FUNCTION_BLOCK PUBLIC DT_TO_TestSuite EXTENDS TcUnit.FB_TestSuite
VAR
END_VAR

Check_DT_TO_BOOL_Max();
Check_DT_TO_BOOL_Min();
Check_DT_TO_BYTE_Max();
Check_DT_TO_BYTE_Min();
Check_DT_TO_BYTE_TooHigh();
Check_DT_TO_WORD_Max();
Check_DT_TO_WORD_Min();
Check_DT_TO_WORD_TooHigh();
Check_DT_TO_DWORD_Max();
Check_DT_TO_DWORD_Min();
Check_DT_TO_LWORD_Max();
Check_DT_TO_LWORD_Min();
Check_DT_TO_SINT_Max();
Check_DT_TO_SINT_Min();
Check_DT_TO_SINT_TooHigh();
Check_DT_TO_INT_Max();
Check_DT_TO_INT_Min();
Check_DT_TO_INT_TooHigh();
Check_DT_TO_DINT_Max();
Check_DT_TO_DINT_Min();
Check_DT_TO_DINT_TooHigh();
Check_DT_TO_LINT_Max();
Check_DT_TO_LINT_Min();
Check_DT_TO_USINT_Max();
Check_DT_TO_USINT_Min();
Check_DT_TO_USINT_TooHigh();
Check_DT_TO_UINT_Max();
Check_DT_TO_UINT_Min();
Check_DT_TO_UINT_TooHigh();
Check_DT_TO_UDINT_Max();
Check_DT_TO_UDINT_Min();
Check_DT_TO_ULINT_Max();
Check_DT_TO_ULINT_Min();
Check_DT_TO_REAL_Max();
Check_DT_TO_REAL_Min();
Check_DT_TO_LREAL_Max();
Check_DT_TO_LREAL_Min();
Check_DT_TO_TIME_Max();
Check_DT_TO_TIME_Min();
Check_DT_TO_TIME_TooHigh();
Check_DT_TO_TOD_Max();
Check_DT_TO_TOD_Min();
Check_DT_TO_TOD_TooHigh();
Check_DT_TO_DATE_Max();
Check_DT_TO_DATE_Min();
Check_DT_TO_DT_Max();
Check_DT_TO_DT_Min();
Check_DT_TO_STRING_Max();
Check_DT_TO_STRING_Min();

METHOD PUBLIC Check_DT_TO_BOOL_Min
VAR
	value : DT := DatatypeLimits.DT_MIN_VALUE;
	actual : BOOL;
	converted : BOOL;
	equal : BOOL;
END_VAR
TEST('Check_DT_TO_BOOL_Min');

// @TEST-RUN
converted := TryConvert_DT_TO_Destination(value, actual);
equal := actual = DT_TO_BOOL(value);

// @TEST-ASSERT
AssertTrue(Condition := equal, Message := 'Did not convert DT to BOOL correctly');
AssertTrue(Condition := converted, Message := 'Did not report DT to BOOL conversion was successful');

TEST_FINISHED();
END_METHOD

METHOD PUBLIC Check_DT_TO_BOOL_Max
VAR
	value : DT := DatatypeLimits.DT_MAX_VALUE;
	actual : BOOL;
	converted : BOOL;
	equal : BOOL;
END_VAR
TEST('Check_DT_TO_BOOL_Max');

// @TEST-RUN
converted := TryConvert_DT_TO_Destination(value, actual);
equal := actual = DT_TO_BOOL(value);

// @TEST-ASSERT
AssertTrue(Condition := equal, Message := 'Did not convert DT to BOOL correctly');
AssertTrue(Condition := converted, Message := 'Did not report DT to BOOL conversion was successful');

TEST_FINISHED();
END_METHOD

METHOD PUBLIC Check_DT_TO_BYTE_Min
VAR
	value : DT := DatatypeLimits.DT_MIN_VALUE;
	actual : BYTE;
	converted : BOOL;
	equal : BOOL;
END_VAR
TEST('Check_DT_TO_BYTE_Min');

// @TEST-RUN
converted := TryConvert_DT_TO_Destination(value, actual);
equal := actual = DT_TO_BYTE(value);

// @TEST-ASSERT
AssertTrue(Condition := equal, Message := 'Did not convert DT to BYTE correctly');
AssertTrue(Condition := converted, Message := 'Did not report DT to BYTE conversion was successful');

TEST_FINISHED();
END_METHOD

METHOD PUBLIC Check_DT_TO_BYTE_TooHigh
VAR
	value : DT := DatatypeLimits.DT_MAX_VALUE;
	actual : BYTE;
	converted : BOOL;
END_VAR
TEST('Check_DT_TO_BYTE_TooHigh');

// @TEST-RUN
converted := TryConvert_DT_TO_Destination(value, actual);

// @TEST-ASSERT
AssertFalse(Condition := converted, Message := 'Did not report DT to BYTE conversion was prevented');

TEST_FINISHED();
END_METHOD

METHOD PUBLIC Check_DT_TO_BYTE_Max
VAR
	value : DT := DatatypeLimits.MAX_VALUE_OF_DT_WHICH_CAN_BE_HELD_IN_A_BYTE;
	actual : BYTE;
	converted : BOOL;
	equal : BOOL;
END_VAR
TEST('Check_DT_TO_BYTE_Max');

// @TEST-RUN
converted := TryConvert_DT_TO_Destination(value, actual);
equal := actual = DT_TO_BYTE(value);

// @TEST-ASSERT
AssertTrue(Condition := equal, Message := 'Did not convert DT to BYTE correctly');
AssertTrue(Condition := converted, Message := 'Did not report DT to BYTE conversion was successful');

TEST_FINISHED();
END_METHOD

METHOD PUBLIC Check_DT_TO_DATE_Min
VAR
	value : DT := DatatypeLimits.DT_MIN_VALUE;
	actual : DATE;
	converted : BOOL;
	equal : BOOL;
END_VAR
TEST('Check_DT_TO_DATE_Min');

// @TEST-RUN
converted := TryConvert_DT_TO_Destination(value, actual);
equal := actual = DT_TO_DATE(value);

// @TEST-ASSERT
AssertTrue(Condition := equal, Message := 'Did not convert DT to DATE correctly');
AssertTrue(Condition := converted, Message := 'Did not report DT to DATE conversion was successful');

TEST_FINISHED();
END_METHOD

METHOD PUBLIC Check_DT_TO_DATE_Max
VAR
	value : DT := DatatypeLimits.DT_MAX_VALUE;
	actual : DATE;
	converted : BOOL;
	equal : BOOL;
END_VAR
TEST('Check_DT_TO_DATE_Max');

// @TEST-RUN
converted := TryConvert_DT_TO_Destination(value, actual);
equal := actual = DT_TO_DATE(value);

// @TEST-ASSERT
AssertTrue(Condition := equal, Message := 'Did not convert DT to DATE correctly');
AssertTrue(Condition := converted, Message := 'Did not report DT to DATE conversion was successful');

TEST_FINISHED();
END_METHOD

METHOD PUBLIC Check_DT_TO_DINT_Min
VAR
	value : DT := DatatypeLimits.DT_MIN_VALUE;
	actual : DINT;
	converted : BOOL;
	equal : BOOL;
END_VAR
TEST('Check_DT_TO_DINT_Min');

// @TEST-RUN
converted := TryConvert_DT_TO_Destination(value, actual);
equal := actual = DT_TO_DINT(value);

// @TEST-ASSERT
AssertTrue(Condition := equal, Message := 'Did not convert DT to DINT correctly');
AssertTrue(Condition := converted, Message := 'Did not report DT to DINT conversion was successful');

TEST_FINISHED();
END_METHOD

METHOD PUBLIC Check_DT_TO_DINT_TooHigh
VAR
	value : DT := DatatypeLimits.DT_MAX_VALUE;
	actual : DINT;
	converted : BOOL;
END_VAR
TEST('Check_DT_TO_DINT_TooHigh');

// @TEST-RUN
converted := TryConvert_DT_TO_Destination(value, actual);

// @TEST-ASSERT
AssertFalse(Condition := converted, Message := 'Did not report DT to DINT conversion was prevented');

TEST_FINISHED();
END_METHOD

METHOD PUBLIC Check_DT_TO_DINT_Max
VAR
	value : DT := DatatypeLimits.MAX_VALUE_OF_DT_WHICH_CAN_BE_HELD_IN_A_DINT;
	actual : DINT;
	converted : BOOL;
	equal : BOOL;
END_VAR
TEST('Check_DT_TO_DINT_Max');

// @TEST-RUN
converted := TryConvert_DT_TO_Destination(value, actual);
equal := actual = DT_TO_DINT(value);

// @TEST-ASSERT
AssertTrue(Condition := equal, Message := 'Did not convert DT to DINT correctly');
AssertTrue(Condition := converted, Message := 'Did not report DT to DINT conversion was successful');

TEST_FINISHED();
END_METHOD

METHOD PUBLIC Check_DT_TO_DT_Min
VAR
	value : DT := DatatypeLimits.DT_MIN_VALUE;
	actual : DT;
	converted : BOOL;
	equal : BOOL;
END_VAR
TEST('Check_DT_TO_DT_Min');

// @TEST-RUN
converted := TryConvert_DT_TO_Destination(value, actual);
equal := actual = value;

// @TEST-ASSERT
AssertTrue(Condition := equal, Message := 'Did not convert DT to DT correctly');
AssertTrue(Condition := converted, Message := 'Did not report DT to DT conversion was successful');

TEST_FINISHED();
END_METHOD

METHOD PUBLIC Check_DT_TO_DT_Max
VAR
	value : DT := DatatypeLimits.DT_MAX_VALUE;
	actual : DT;
	converted : BOOL;
	equal : BOOL;
END_VAR
TEST('Check_DT_TO_DT_Max');

// @TEST-RUN
converted := TryConvert_DT_TO_Destination(value, actual);
equal := actual = value;

// @TEST-ASSERT
AssertTrue(Condition := equal, Message := 'Did not convert DT to DT correctly');
AssertTrue(Condition := converted, Message := 'Did not report DT to DT conversion was successful');

TEST_FINISHED();
END_METHOD

METHOD PUBLIC Check_DT_TO_DWORD_Min
VAR
	value : DT := DatatypeLimits.DT_MIN_VALUE;
	actual : DWORD;
	converted : BOOL;
	equal : BOOL;
END_VAR
TEST('Check_DT_TO_DWORD_Min');

// @TEST-RUN
converted := TryConvert_DT_TO_Destination(value, actual);
equal := actual = DT_TO_DWORD(value);

// @TEST-ASSERT
AssertTrue(Condition := equal, Message := 'Did not convert DT to DWORD correctly');
AssertTrue(Condition := converted, Message := 'Did not report DT to DWORD conversion was successful');

TEST_FINISHED();
END_METHOD

METHOD PUBLIC Check_DT_TO_DWORD_Max
VAR
	value : DT := DatatypeLimits.DT_MAX_VALUE;
	actual : DWORD;
	converted : BOOL;
	equal : BOOL;
END_VAR
TEST('Check_DT_TO_DWORD_Max');

// @TEST-RUN
converted := TryConvert_DT_TO_Destination(value, actual);
equal := actual = DT_TO_DWORD(value);

// @TEST-ASSERT
AssertTrue(Condition := equal, Message := 'Did not convert DT to DWORD correctly');
AssertTrue(Condition := converted, Message := 'Did not report DT to DWORD conversion was successful');

TEST_FINISHED();
END_METHOD

METHOD PUBLIC Check_DT_TO_INT_Min
VAR
	value : DT := DatatypeLimits.DT_MIN_VALUE;
	actual : INT;
	converted : BOOL;
	equal : BOOL;
END_VAR
TEST('Check_DT_TO_INT_Min');

// @TEST-RUN
converted := TryConvert_DT_TO_Destination(value, actual);
equal := actual = DT_TO_INT(value);

// @TEST-ASSERT
AssertTrue(Condition := equal, Message := 'Did not convert DT to INT correctly');
AssertTrue(Condition := converted, Message := 'Did not report DT to INT conversion was successful');

TEST_FINISHED();
END_METHOD

METHOD PUBLIC Check_DT_TO_INT_TooHigh
VAR
	value : DT := DatatypeLimits.DT_MAX_VALUE;
	actual : INT;
	converted : BOOL;
END_VAR
TEST('Check_DT_TO_INT_TooHigh');

// @TEST-RUN
converted := TryConvert_DT_TO_Destination(value, actual);

// @TEST-ASSERT
AssertFalse(Condition := converted, Message := 'Did not report DT to INT conversion was prevented');

TEST_FINISHED();
END_METHOD

METHOD PUBLIC Check_DT_TO_INT_Max
VAR
	value : DT := DatatypeLimits.MAX_VALUE_OF_DT_WHICH_CAN_BE_HELD_IN_A_INT;
	actual : INT;
	converted : BOOL;
	equal : BOOL;
END_VAR
TEST('Check_DT_TO_INT_Max');

// @TEST-RUN
converted := TryConvert_DT_TO_Destination(value, actual);
equal := actual = DT_TO_INT(value);

// @TEST-ASSERT
AssertTrue(Condition := equal, Message := 'Did not convert DT to INT correctly');
AssertTrue(Condition := converted, Message := 'Did not report DT to INT conversion was successful');

TEST_FINISHED();
END_METHOD

METHOD PUBLIC Check_DT_TO_LINT_Min
VAR
	value : DT := DatatypeLimits.DT_MIN_VALUE;
	actual : LINT;
	converted : BOOL;
	equal : BOOL;
END_VAR
TEST('Check_DT_TO_LINT_Min');

// @TEST-RUN
converted := TryConvert_DT_TO_Destination(value, actual);
equal := actual = DT_TO_LINT(value);

// @TEST-ASSERT
AssertTrue(Condition := equal, Message := 'Did not convert DT to LINT correctly');
AssertTrue(Condition := converted, Message := 'Did not report DT to LINT conversion was successful');

TEST_FINISHED();
END_METHOD

METHOD PUBLIC Check_DT_TO_LINT_Max
VAR
	value : DT := DatatypeLimits.DT_MAX_VALUE;
	actual : LINT;
	converted : BOOL;
	equal : BOOL;
END_VAR
TEST('Check_DT_TO_LINT_Max');

// @TEST-RUN
converted := TryConvert_DT_TO_Destination(value, actual);
equal := actual = DT_TO_LINT(value);

// @TEST-ASSERT
AssertTrue(Condition := equal, Message := 'Did not convert DT to LINT correctly');
AssertTrue(Condition := converted, Message := 'Did not report DT to LINT conversion was successful');

TEST_FINISHED();
END_METHOD

METHOD PUBLIC Check_DT_TO_LREAL_Min
VAR
	value : DT := DatatypeLimits.DT_MIN_VALUE;
	actual : LREAL;
	converted : BOOL;
	equal : BOOL;
END_VAR
TEST('Check_DT_TO_LREAL_Min');

// @TEST-RUN
converted := TryConvert_DT_TO_Destination(value, actual);
equal := actual = DT_TO_LREAL(value);

// @TEST-ASSERT
AssertTrue(Condition := equal, Message := 'Did not convert DT to LREAL correctly');
AssertTrue(Condition := converted, Message := 'Did not report DT to LREAL conversion was successful');

TEST_FINISHED();
END_METHOD

METHOD PUBLIC Check_DT_TO_LREAL_Max
VAR
	value : DT := DatatypeLimits.DT_MAX_VALUE;
	actual : LREAL;
	converted : BOOL;
	equal : BOOL;
END_VAR
TEST('Check_DT_TO_LREAL_Max');

// @TEST-RUN
converted := TryConvert_DT_TO_Destination(value, actual);
equal := actual = DT_TO_LREAL(value);

// @TEST-ASSERT
AssertTrue(Condition := equal, Message := 'Did not convert DT to LREAL correctly');
AssertTrue(Condition := converted, Message := 'Did not report DT to LREAL conversion was successful');

TEST_FINISHED();
END_METHOD

METHOD PUBLIC Check_DT_TO_LWORD_Min
VAR
	value : DT := DatatypeLimits.DT_MIN_VALUE;
	actual : LWORD;
	converted : BOOL;
	equal : BOOL;
END_VAR
TEST('Check_DT_TO_LWORD_Min');

// @TEST-RUN
converted := TryConvert_DT_TO_Destination(value, actual);
equal := actual = DT_TO_LWORD(value);

// @TEST-ASSERT
AssertTrue(Condition := equal, Message := 'Did not convert DT to LWORD correctly');
AssertTrue(Condition := converted, Message := 'Did not report DT to LWORD conversion was successful');

TEST_FINISHED();
END_METHOD

METHOD PUBLIC Check_DT_TO_LWORD_Max
VAR
	value : DT := DatatypeLimits.DT_MAX_VALUE;
	actual : LWORD;
	converted : BOOL;
	equal : BOOL;
END_VAR
TEST('Check_DT_TO_LWORD_Max');

// @TEST-RUN
converted := TryConvert_DT_TO_Destination(value, actual);
equal := actual = DT_TO_LWORD(value);

// @TEST-ASSERT
AssertTrue(Condition := equal, Message := 'Did not convert DT to LWORD correctly');
AssertTrue(Condition := converted, Message := 'Did not report DT to LWORD conversion was successful');

TEST_FINISHED();
END_METHOD

METHOD PUBLIC Check_DT_TO_REAL_Min
VAR
	value : DT := DatatypeLimits.DT_MIN_VALUE;
	actual : REAL;
	converted : BOOL;
	equal : BOOL;
END_VAR
TEST('Check_DT_TO_REAL_Min');

// @TEST-RUN
converted := TryConvert_DT_TO_Destination(value, actual);
equal := actual = DT_TO_REAL(value);

// @TEST-ASSERT
AssertTrue(Condition := equal, Message := 'Did not convert DT to REAL correctly');
AssertTrue(Condition := converted, Message := 'Did not report DT to REAL conversion was successful');

TEST_FINISHED();
END_METHOD

METHOD PUBLIC Check_DT_TO_REAL_Max
VAR
	value : DT := DatatypeLimits.DT_MAX_VALUE;
	actual : REAL;
	converted : BOOL;
	equal : BOOL;
END_VAR
TEST('Check_DT_TO_REAL_Max');

// @TEST-RUN
converted := TryConvert_DT_TO_Destination(value, actual);
equal := actual = DT_TO_REAL(value);

// @TEST-ASSERT
AssertTrue(Condition := equal, Message := 'Did not convert DT to REAL correctly');
AssertTrue(Condition := converted, Message := 'Did not report DT to REAL conversion was successful');

TEST_FINISHED();
END_METHOD

METHOD PUBLIC Check_DT_TO_SINT_Min
VAR
	value : DT := DatatypeLimits.DT_MIN_VALUE;
	actual : SINT;
	converted : BOOL;
	equal : BOOL;
END_VAR
TEST('Check_DT_TO_SINT_Min');

// @TEST-RUN
converted := TryConvert_DT_TO_Destination(value, actual);
equal := actual = DT_TO_SINT(value);

// @TEST-ASSERT
AssertTrue(Condition := equal, Message := 'Did not convert DT to SINT correctly');
AssertTrue(Condition := converted, Message := 'Did not report DT to SINT conversion was successful');

TEST_FINISHED();
END_METHOD

METHOD PUBLIC Check_DT_TO_SINT_TooHigh
VAR
	value : DT := DatatypeLimits.DT_MAX_VALUE;
	actual : SINT;
	converted : BOOL;
END_VAR
TEST('Check_DT_TO_SINT_TooHigh');

// @TEST-RUN
converted := TryConvert_DT_TO_Destination(value, actual);

// @TEST-ASSERT
AssertFalse(Condition := converted, Message := 'Did not report DT to SINT conversion was prevented');

TEST_FINISHED();
END_METHOD

METHOD PUBLIC Check_DT_TO_SINT_Max
VAR
	value : DT := DatatypeLimits.MAX_VALUE_OF_DT_WHICH_CAN_BE_HELD_IN_A_SINT;
	actual : SINT;
	converted : BOOL;
	equal : BOOL;
END_VAR
TEST('Check_DT_TO_SINT_Max');

// @TEST-RUN
converted := TryConvert_DT_TO_Destination(value, actual);
equal := actual = DT_TO_SINT(value);

// @TEST-ASSERT
AssertTrue(Condition := equal, Message := 'Did not convert DT to SINT correctly');
AssertTrue(Condition := converted, Message := 'Did not report DT to SINT conversion was successful');

TEST_FINISHED();
END_METHOD

METHOD PUBLIC Check_DT_TO_STRING_Min
VAR
	value : DT := DatatypeLimits.DT_MIN_VALUE;
	actual : STRING;
	converted : BOOL;
	equal : BOOL;
END_VAR
TEST('Check_DT_TO_STRING_Min');

// @TEST-RUN
converted := TryConvert_DT_TO_Destination(value, actual);
equal := actual = DT_TO_STRING(value);

// @TEST-ASSERT
AssertTrue(Condition := equal, Message := 'Did not convert DT to STRING correctly');
AssertTrue(Condition := converted, Message := 'Did not report DT to STRING conversion was successful');

TEST_FINISHED();
END_METHOD

METHOD PUBLIC Check_DT_TO_STRING_Max
VAR
	value : DT := DatatypeLimits.DT_MAX_VALUE;
	actual : STRING;
	converted : BOOL;
	equal : BOOL;
END_VAR
TEST('Check_DT_TO_STRING_Max');

// @TEST-RUN
converted := TryConvert_DT_TO_Destination(value, actual);
equal := actual = DT_TO_STRING(value);

// @TEST-ASSERT
AssertTrue(Condition := equal, Message := 'Did not convert DT to STRING correctly');
AssertTrue(Condition := converted, Message := 'Did not report DT to STRING conversion was successful');

TEST_FINISHED();
END_METHOD

METHOD PUBLIC Check_DT_TO_TIME_Min
VAR
	value : DT := DatatypeLimits.DT_MIN_VALUE;
	actual : TIME;
	converted : BOOL;
	equal : BOOL;
END_VAR
TEST('Check_DT_TO_TIME_Min');

// @TEST-RUN
converted := TryConvert_DT_TO_Destination(value, actual);
equal := actual = DT_TO_TIME(value);

// @TEST-ASSERT
AssertTrue(Condition := equal, Message := 'Did not convert DT to TIME correctly');
AssertTrue(Condition := converted, Message := 'Did not report DT to TIME conversion was successful');

TEST_FINISHED();
END_METHOD

METHOD PUBLIC Check_DT_TO_TIME_TooHigh
VAR
	value : DT := DatatypeLimits.DT_MAX_VALUE;
	actual : TIME;
	converted : BOOL;
END_VAR
TEST('Check_DT_TO_TIME_TooHigh');

// @TEST-RUN
converted := TryConvert_DT_TO_Destination(value, actual);

// @TEST-ASSERT
AssertFalse(Condition := converted, Message := 'Did not report DT to TIME conversion was prevented');

TEST_FINISHED();
END_METHOD

METHOD PUBLIC Check_DT_TO_TIME_Max
VAR
	value : DT := DatatypeLimits.MAX_VALUE_OF_DT_WHICH_CAN_BE_HELD_IN_A_TIME;
	actual : TIME;
	converted : BOOL;
	equal : BOOL;
END_VAR
TEST('Check_DT_TO_TIME_Max');

// @TEST-RUN
converted := TryConvert_DT_TO_Destination(value, actual);
equal := actual = DT_TO_TIME(value);

// @TEST-ASSERT
AssertTrue(Condition := equal, Message := 'Did not convert DT to TIME correctly');
AssertTrue(Condition := converted, Message := 'Did not report DT to TIME conversion was successful');

TEST_FINISHED();
END_METHOD

METHOD PUBLIC Check_DT_TO_TOD_Min
VAR
	value : DT := DatatypeLimits.DT_MIN_VALUE;
	actual : TOD;
	converted : BOOL;
	equal : BOOL;
END_VAR
TEST('Check_DT_TO_TOD_Min');

// @TEST-RUN
converted := TryConvert_DT_TO_Destination(value, actual);
equal := actual = DT_TO_TOD(value);

// @TEST-ASSERT
AssertTrue(Condition := equal, Message := 'Did not convert DT to TOD correctly');
AssertTrue(Condition := converted, Message := 'Did not report DT to TOD conversion was successful');

TEST_FINISHED();
END_METHOD

METHOD PUBLIC Check_DT_TO_TOD_TooHigh
VAR
	value : DT := DatatypeLimits.DT_MAX_VALUE;
	actual : TOD;
	converted : BOOL;
END_VAR
TEST('Check_DT_TO_TOD_TooHigh');

// @TEST-RUN
converted := TryConvert_DT_TO_Destination(value, actual);

// @TEST-ASSERT
AssertFalse(Condition := converted, Message := 'Did not report DT to TOD conversion was prevented');

TEST_FINISHED();
END_METHOD

METHOD PUBLIC Check_DT_TO_TOD_Max
VAR
	value : DT := DatatypeLimits.MAX_VALUE_OF_DT_WHICH_CAN_BE_HELD_IN_A_TOD;
	actual : TOD;
	converted : BOOL;
	equal : BOOL;
END_VAR
TEST('Check_DT_TO_TOD_Max');

// @TEST-RUN
converted := TryConvert_DT_TO_Destination(value, actual);
equal := actual = DT_TO_TOD(value);

// @TEST-ASSERT
AssertTrue(Condition := equal, Message := 'Did not convert DT to TOD correctly');
AssertTrue(Condition := converted, Message := 'Did not report DT to TOD conversion was successful');

TEST_FINISHED();
END_METHOD

METHOD PUBLIC Check_DT_TO_UDINT_Min
VAR
	value : DT := DatatypeLimits.DT_MIN_VALUE;
	actual : UDINT;
	converted : BOOL;
	equal : BOOL;
END_VAR
TEST('Check_DT_TO_UDINT_Min');

// @TEST-RUN
converted := TryConvert_DT_TO_Destination(value, actual);
equal := actual = DT_TO_UDINT(value);

// @TEST-ASSERT
AssertTrue(Condition := equal, Message := 'Did not convert DT to UDINT correctly');
AssertTrue(Condition := converted, Message := 'Did not report DT to UDINT conversion was successful');

TEST_FINISHED();
END_METHOD

METHOD PUBLIC Check_DT_TO_UDINT_Max
VAR
	value : DT := DatatypeLimits.DT_MAX_VALUE;
	actual : UDINT;
	converted : BOOL;
	equal : BOOL;
END_VAR
TEST('Check_DT_TO_UDINT_Max');

// @TEST-RUN
converted := TryConvert_DT_TO_Destination(value, actual);
equal := actual = DT_TO_UDINT(value);

// @TEST-ASSERT
AssertTrue(Condition := equal, Message := 'Did not convert DT to UDINT correctly');
AssertTrue(Condition := converted, Message := 'Did not report DT to UDINT conversion was successful');

TEST_FINISHED();
END_METHOD

METHOD PUBLIC Check_DT_TO_UINT_Min
VAR
	value : DT := DatatypeLimits.DT_MIN_VALUE;
	actual : UINT;
	converted : BOOL;
	equal : BOOL;
END_VAR
TEST('Check_DT_TO_UINT_Min');

// @TEST-RUN
converted := TryConvert_DT_TO_Destination(value, actual);
equal := actual = DT_TO_UINT(value);

// @TEST-ASSERT
AssertTrue(Condition := equal, Message := 'Did not convert DT to UINT correctly');
AssertTrue(Condition := converted, Message := 'Did not report DT to UINT conversion was successful');

TEST_FINISHED();
END_METHOD

METHOD PUBLIC Check_DT_TO_UINT_TooHigh
VAR
	value : DT := DatatypeLimits.DT_MAX_VALUE;
	actual : UINT;
	converted : BOOL;
END_VAR
TEST('Check_DT_TO_UINT_TooHigh');

// @TEST-RUN
converted := TryConvert_DT_TO_Destination(value, actual);

// @TEST-ASSERT
AssertFalse(Condition := converted, Message := 'Did not report DT to UINT conversion was prevented');

TEST_FINISHED();
END_METHOD

METHOD PUBLIC Check_DT_TO_UINT_Max
VAR
	value : DT := DatatypeLimits.MAX_VALUE_OF_DT_WHICH_CAN_BE_HELD_IN_A_UINT;
	actual : UINT;
	converted : BOOL;
	equal : BOOL;
END_VAR
TEST('Check_DT_TO_UINT_Max');

// @TEST-RUN
converted := TryConvert_DT_TO_Destination(value, actual);
equal := actual = DT_TO_UINT(value);

// @TEST-ASSERT
AssertTrue(Condition := equal, Message := 'Did not convert DT to UINT correctly');
AssertTrue(Condition := converted, Message := 'Did not report DT to UINT conversion was successful');

TEST_FINISHED();
END_METHOD

METHOD PUBLIC Check_DT_TO_ULINT_Min
VAR
	value : DT := DatatypeLimits.DT_MIN_VALUE;
	actual : ULINT;
	converted : BOOL;
	equal : BOOL;
END_VAR
TEST('Check_DT_TO_ULINT_Min');

// @TEST-RUN
converted := TryConvert_DT_TO_Destination(value, actual);
equal := actual = DT_TO_ULINT(value);

// @TEST-ASSERT
AssertTrue(Condition := equal, Message := 'Did not convert DT to ULINT correctly');
AssertTrue(Condition := converted, Message := 'Did not report DT to ULINT conversion was successful');

TEST_FINISHED();
END_METHOD

METHOD PUBLIC Check_DT_TO_ULINT_Max
VAR
	value : DT := DatatypeLimits.DT_MAX_VALUE;
	actual : ULINT;
	converted : BOOL;
	equal : BOOL;
END_VAR
TEST('Check_DT_TO_ULINT_Max');

// @TEST-RUN
converted := TryConvert_DT_TO_Destination(value, actual);
equal := actual = DT_TO_ULINT(value);

// @TEST-ASSERT
AssertTrue(Condition := equal, Message := 'Did not convert DT to ULINT correctly');
AssertTrue(Condition := converted, Message := 'Did not report DT to ULINT conversion was successful');

TEST_FINISHED();
END_METHOD

METHOD PUBLIC Check_DT_TO_USINT_Min
VAR
	value : DT := DatatypeLimits.DT_MIN_VALUE;
	actual : USINT;
	converted : BOOL;
	equal : BOOL;
END_VAR
TEST('Check_DT_TO_USINT_Min');

// @TEST-RUN
converted := TryConvert_DT_TO_Destination(value, actual);
equal := actual = DT_TO_USINT(value);

// @TEST-ASSERT
AssertTrue(Condition := equal, Message := 'Did not convert DT to USINT correctly');
AssertTrue(Condition := converted, Message := 'Did not report DT to USINT conversion was successful');

TEST_FINISHED();
END_METHOD

METHOD PUBLIC Check_DT_TO_USINT_TooHigh
VAR
	value : DT := DatatypeLimits.DT_MAX_VALUE;
	actual : USINT;
	converted : BOOL;
END_VAR
TEST('Check_DT_TO_USINT_TooHigh');

// @TEST-RUN
converted := TryConvert_DT_TO_Destination(value, actual);

// @TEST-ASSERT
AssertFalse(Condition := converted, Message := 'Did not report DT to USINT conversion was prevented');

TEST_FINISHED();
END_METHOD

METHOD PUBLIC Check_DT_TO_USINT_Max
VAR
	value : DT := DatatypeLimits.MAX_VALUE_OF_DT_WHICH_CAN_BE_HELD_IN_A_USINT;
	actual : USINT;
	converted : BOOL;
	equal : BOOL;
END_VAR
TEST('Check_DT_TO_USINT_Max');

// @TEST-RUN
converted := TryConvert_DT_TO_Destination(value, actual);
equal := actual = DT_TO_USINT(value);

// @TEST-ASSERT
AssertTrue(Condition := equal, Message := 'Did not convert DT to USINT correctly');
AssertTrue(Condition := converted, Message := 'Did not report DT to USINT conversion was successful');

TEST_FINISHED();
END_METHOD

METHOD PUBLIC Check_DT_TO_WORD_Min
VAR
	value : DT := DatatypeLimits.DT_MIN_VALUE;
	actual : WORD;
	converted : BOOL;
	equal : BOOL;
END_VAR
TEST('Check_DT_TO_WORD_Min');

// @TEST-RUN
converted := TryConvert_DT_TO_Destination(value, actual);
equal := actual = DT_TO_WORD(value);

// @TEST-ASSERT
AssertTrue(Condition := equal, Message := 'Did not convert DT to WORD correctly');
AssertTrue(Condition := converted, Message := 'Did not report DT to WORD conversion was successful');

TEST_FINISHED();
END_METHOD

METHOD PUBLIC Check_DT_TO_WORD_TooHigh
VAR
	value : DT := DatatypeLimits.DT_MAX_VALUE;
	actual : WORD;
	converted : BOOL;
END_VAR
TEST('Check_DT_TO_WORD_TooHigh');

// @TEST-RUN
converted := TryConvert_DT_TO_Destination(value, actual);

// @TEST-ASSERT
AssertFalse(Condition := converted, Message := 'Did not report DT to WORD conversion was prevented');

TEST_FINISHED();
END_METHOD

METHOD PUBLIC Check_DT_TO_WORD_Max
VAR
	value : DT := DatatypeLimits.MAX_VALUE_OF_DT_WHICH_CAN_BE_HELD_IN_A_WORD;
	actual : WORD;
	converted : BOOL;
	equal : BOOL;
END_VAR
TEST('Check_DT_TO_WORD_Max');

// @TEST-RUN
converted := TryConvert_DT_TO_Destination(value, actual);
equal := actual = DT_TO_WORD(value);

// @TEST-ASSERT
AssertTrue(Condition := equal, Message := 'Did not convert DT to WORD correctly');
AssertTrue(Condition := converted, Message := 'Did not report DT to WORD conversion was successful');

TEST_FINISHED();
END_METHOD

END_FUNCTION_BLOCK

(* stored: Version 1.1.0.1, ProductVersion 3.1.4024.12
   POU DT_TO_TestSuite: Id {bf7dd3c3-a216-4f6d-b55b-d7ed22da8d01}, SpecialFunc None
   Method Check_DT_TO_BOOL_Min: Id {5f8470c0-2c79-4f55-871d-26ad725fa846}
   Method Check_DT_TO_BOOL_Max: Id {5bdea242-6595-4bca-98b6-2cddab1d1f72}
   Method Check_DT_TO_BYTE_Min: Id {06fcbc49-f6d4-4351-9177-ff19f5f11ed6}
   Method Check_DT_TO_BYTE_TooHigh: Id {8129c381-b2b8-4631-920c-865d12d1b852}
   Method Check_DT_TO_BYTE_Max: Id {ac7a9973-cf3b-45e8-9747-1b349070cec5}
   Method Check_DT_TO_DATE_Min: Id {226886ae-190e-4c60-b37b-6c0f66452a68}
   Method Check_DT_TO_DATE_Max: Id {eb6ae078-bf9a-4ccb-aee8-08df166073ab}
   Method Check_DT_TO_DINT_Min: Id {ab7c729b-9a4e-4fd6-b290-050b0be427f2}
   Method Check_DT_TO_DINT_TooHigh: Id {b8295118-f387-4993-91fd-10707ff00abc}
   Method Check_DT_TO_DINT_Max: Id {cc58d98a-2e63-4d35-b6f9-3c107731d675}
   Method Check_DT_TO_DT_Min: Id {4cabeb14-8f46-4346-b1e3-a6fd6e0e03c1}
   Method Check_DT_TO_DT_Max: Id {459f9ccb-fc9a-4393-a1a6-4ef136fed25e}
   Method Check_DT_TO_DWORD_Min: Id {78683698-3c33-47ec-a5c3-561e6327e867}
   Method Check_DT_TO_DWORD_Max: Id {c68b567a-ad66-4f9a-9f97-3663c6d100b5}
   Method Check_DT_TO_INT_Min: Id {2a6e1706-89f1-47b6-8394-9668593d0377}
   Method Check_DT_TO_INT_TooHigh: Id {f44d661c-18a0-4dc2-8ccc-b318a72834b3}
   Method Check_DT_TO_INT_Max: Id {c834fcf7-66ac-4cfd-a41a-190257b7ee5a}
   Method Check_DT_TO_LINT_Min: Id {d4bf5445-7888-41ee-8d11-c40f9565d6ca}
   Method Check_DT_TO_LINT_Max: Id {0a2de31c-49c1-4f25-8008-68220e008e37}
   Method Check_DT_TO_LREAL_Min: Id {680015b1-3277-4a3e-a294-cd7b2a2b0c66}
   Method Check_DT_TO_LREAL_Max: Id {df0641a2-7bc9-4773-86df-6b979a18cf48}
   Method Check_DT_TO_LWORD_Min: Id {0cef231d-dc62-4838-8856-88cae25dc627}
   Method Check_DT_TO_LWORD_Max: Id {1cf5e99c-93f7-477f-ac77-4ce1e2c6e5d2}
   Method Check_DT_TO_REAL_Min: Id {25000aa5-c5c3-439e-8b59-c18266b59912}
   Method Check_DT_TO_REAL_Max: Id {700da25b-dcad-4d3a-b779-3ccca65029fc}
   Method Check_DT_TO_SINT_Min: Id {f935d357-512e-4d01-88b5-509233c2f7b5}
   Method Check_DT_TO_SINT_TooHigh: Id {71b2eabc-c377-48ee-ae64-00a0460a77f0}
   Method Check_DT_TO_SINT_Max: Id {c5c531bf-44ac-4328-a661-a1ee73ce6345}
   Method Check_DT_TO_STRING_Min: Id {1cea9b03-2996-472e-9ed2-49fb1b292a1f}
   Method Check_DT_TO_STRING_Max: Id {dcba52b5-9d18-4e52-aa76-22ed4956e459}
   Method Check_DT_TO_TIME_Min: Id {968517ae-e311-4153-8939-8ce6d96e86ce}
   Method Check_DT_TO_TIME_TooHigh: Id {452df00a-2f25-4e75-949c-69ed3bdb9119}
   Method Check_DT_TO_TIME_Max: Id {c4cc77ff-ecc1-4801-81ac-09ad9274883f}
   Method Check_DT_TO_TOD_Min: Id {0e0f8924-353d-40b7-b3c4-6ba2f821078e}
   Method Check_DT_TO_TOD_TooHigh: Id {b5876a20-dda6-42dc-9915-bce7eb88a552}
   Method Check_DT_TO_TOD_Max: Id {32befd99-5da8-4871-8b49-c492674e74a6}
   Method Check_DT_TO_UDINT_Min: Id {498e6f5f-7681-4cde-b4e6-3052f3ef81e8}
   Method Check_DT_TO_UDINT_Max: Id {038d096a-032f-44a0-8248-2d5e027b4078}
   Method Check_DT_TO_UINT_Min: Id {62368b26-fb85-44ca-94db-bc475b90cfc7}
   Method Check_DT_TO_UINT_TooHigh: Id {d4703453-babe-4c8d-be75-30b2ff2288bb}
   Method Check_DT_TO_UINT_Max: Id {992dd180-7cc0-4041-a806-debbf34af8c2}
   Method Check_DT_TO_ULINT_Min: Id {0028fb3c-45cd-4ac5-ab3e-a64846cf8533}
   Method Check_DT_TO_ULINT_Max: Id {dda6dd33-0447-4be6-8c02-56bbc7663940}
   Method Check_DT_TO_USINT_Min: Id {c76b0680-8e1b-46e7-a655-0458e7d6c691}
   Method Check_DT_TO_USINT_TooHigh: Id {472ed588-62f6-43a1-be22-bd8af3d50995}
   Method Check_DT_TO_USINT_Max: Id {41c0374b-4a50-45cd-b698-6c4c92a767b8}
   Method Check_DT_TO_WORD_Min: Id {a4f84542-6e1b-4f73-ac77-510efb6ab5fd}
   Method Check_DT_TO_WORD_TooHigh: Id {16afbe70-12e7-4a74-9521-87e308d48206}
   Method Check_DT_TO_WORD_Max: Id {e44543d1-dc63-4b7d-b261-aeae98ac360d} *)
